// TIA Portal V17 export
// export: Created 2023-05-07T12:12:22.6858465Z, ExportSetting WithDefaults, DisplayName Totally Integrated Automation Portal, DisplayVersion V17, DisplayName TIA Portal Openness, DisplayVersion V17, DisplayName TIA Portal Version Control Interface, DisplayVersion V17, DisplayName TIA Portal Test Suite Advanced, DisplayVersion V17, DisplayName STEP 7 Professional, DisplayVersion V17, DisplayName SIMATIC Energy Suite, DisplayVersion V17, DisplayName STEP 7 Safety, DisplayVersion V17, DisplayName WinCC Professional, DisplayVersion V17
DATA_BLOCK "StartStop_DB"   // DB19
VERSION : 0.1
// stored: AutoNumber true, InstanceOfName StartStop, InstanceOfType FB
"StartStop"
   // VAR_INPUT
   //    Start : Bool;
   //    Stop : Bool;
   // END_VAR
   // VAR_OUTPUT
   //    Q : Bool;
   // END_VAR
   // VAR
   //    statSR : Bool;
   //    statRisEdge : Bool;
   // END_VAR
BEGIN
END_DATA_BLOCK
